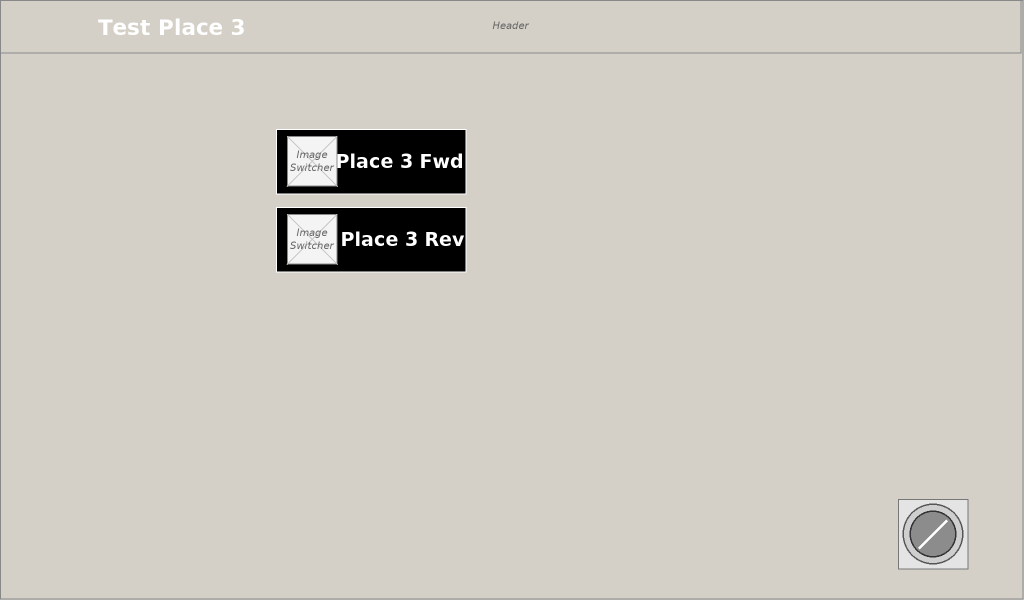
VISUALIZATION Test_Place3  // 1024x600
    Frame (0,-2 1021x55)
        shows Header()
    Label (95,15 250x25), "Test Place 3"
    RotarySwitch (898,499 70x70), variable: HMI_GVL.bTestModeEnablePlacing3, behaviour: TOGGLE, style: Switch-RotarySwitch-Gray
    RoundedRectangle (276,129 190x65)
        toggle Status_GVL.stMotor_Placing3.iTestForward
    Label (331,149 137x25), "Place 3 Fwd"
    ImageSwitcher (287,136 50x50), variable: Status_GVL.stMotor_Placing3.iTestForward, behaviour: TOGGLE
    RoundedRectangle (276,207 190x65)
        toggle Status_GVL.stMotor_Placing3.iTestReverse
    Label (334,227 137x25), "Place 3 Rev"
    ImageSwitcher (287,214 50x50), variable: Status_GVL.stMotor_Placing3.iTestReverse, behaviour: TOGGLE
END_VISUALIZATION

(* stored: Version 1.1.0.1, ProductVersion 3.1.4024.12
   Visu Test_Place3: Id {ad637eda-1d8c-4847-8314-d5c54b41fc4d} *)
